(* CODESYS project mpm_fbresult.library
   Title: MPM_FBResult
   Version: 0.0.1.5
   Placeholder: MPM_FBResult
   Company: MatrixPM

Project tree, tasks and I/O mapping:
  data type E_Result
  function block FB_Result_Base [ST]: M_Excute_Ex, M_Execute
  function block FB_ResultBaseITF [ST]: M_Excute_Ex, P_itfResultEx
  function block FB_ResultHelper [ST]: M_MethodResult, P_Result
  function block FB_ResultHelper_V2 [ST]: M_MethodResult
  function block FB_ResultHelper_V2_1 [ST]: M_MethodResult, P_MethodResult
  function block FB_Templete [ST]: M_Execute
  function block FB_Templete_V2 [ST]: M_Execute
  interface ITF_Result: M_Execute
  interface ITF_ResultExtended: _M_Excute
*)

// E_Result
{attribute 'qualified_only'}
TYPE E_Result :
(
	S_OK := 0,
	S_DONE := 1,
	S_FAILED := -1,
	S_WORKING := 3
)DINT;
END_TYPE

// FB_Result_Base
FUNCTION_BLOCK ABSTRACT FB_Result_Base EXTENDS FB_ResultHelper IMPLEMENTS ITF_Result //used to added HRresult to a FB. 
VAR_INPUT
END_VAR
VAR_OUTPUT
END_VAR
VAR
END_VAR

METHOD PROTECTED ABSTRACT M_Excute_Ex : DINT
VAR_INPUT
	lastResult	: DINT;
END_VAR
VAR_INST
END_VAR
END_METHOD

{warning 'add method implementation '}
METHOD FINAL M_Execute : DINT
VAR_INPUT
	lastResult	: DINT;
END_VAR
IF M_MethodResult(M_Execute,lastResult := lastResult) = FALSE THEN
	RETURN;
ELSE
	THIS^.P_Result := THIS^.M_Excute_Ex(THIS^.P_Result);	//FBs implementation
END_IF
END_METHOD

END_FUNCTION_BLOCK

// FB_ResultHelper
(*
Used to implement HRResult style programing to a meathod. This should be implemented inside of a meathod in VAR_INST becuase
this holds state. This should only be used if the meathod won't be able to return the final result in one scan. (async)
*)
FUNCTION_BLOCK FB_ResultHelper //Used to implement HRResult style programing to a meathod. 
VAR_INPUT
END_VAR
VAR_OUTPUT
END_VAR
VAR
	_lastResult			: DINT;		
	pMethodResult		: REFERENCE TO DINT;		
END_VAR
VAR_TEMP
	
END_VAR

METHOD PUBLIC FINAL M_MethodResult : BOOL
VAR_INPUT
	meathodResultRef	: REFERENCE TO DINT;
	lastResult			: DINT;
END_VAR
VAR
END_VAR
VAR_OUTPUT
END_VAR
VAR_INST
END_VAR
IF ADR(meathodResultRef) = 0 THEN
	M_MethodResult := FALSE;	
ELSIF (lastResult > 0 AND (_lastResult = 0 OR _lastResult <> lastResult)) OR ABS(lastResult) = 1 THEN
	meathodResultRef := lastResult;
	M_MethodResult := FALSE;	
ELSIF lastResult = 0 THEN
	pMethodResult REF= meathodResultRef;
	_lastResult := 0;
	M_MethodResult := TRUE;		
ELSE
	pMethodResult REF= meathodResultRef;
	pMethodResult := lastResult;
	M_MethodResult := TRUE;
	_lastResult := lastResult;
END_IF
END_METHOD

PROPERTY PUBLIC P_Result : DINT
GET
IF ADR(pMethodResult) > 0 THEN
	P_Result := pMethodResult;
ELSE
	P_Result := -1; //Maybe 1?
END_IF
END_GET
SET
IF ADR(pMethodResult) > 0 THEN
	_lastResult := P_Result;
	pMethodResult := P_Result;
END_IF
END_SET
END_PROPERTY

END_FUNCTION_BLOCK

// ITF_Result
INTERFACE ITF_Result

METHOD M_Execute : DINT
VAR_INPUT
	lastResult			: DINT;
END_VAR
END_METHOD

END_INTERFACE

// FB_ResultBaseITF
FUNCTION_BLOCK FB_ResultBaseITF EXTENDS FB_Result_Base //used for librays that I can't extened. 
VAR_INPUT
END_VAR
VAR_OUTPUT
END_VAR
VAR
	itfResultEx	: ITF_ResultExtended;
END_VAR

METHOD PROTECTED FINAL M_Excute_Ex : DINT
VAR_INPUT
	lastResult	: DINT;
END_VAR
VAR_INST
END_VAR
IF ADR(itfResultEx) = 0 THEN
	M_Excute_Ex := 1;
	RETURN; 
ELSE
	M_Excute_Ex := itfResultEx._M_Excute(lastResult);
	RETURN; 	
END_IF
END_METHOD

PROPERTY PUBLIC P_itfResultEx : ITF_ResultExtended // has to be set every cycle.
SET
itfResultEx := P_itfResultEx;
END_SET
END_PROPERTY

END_FUNCTION_BLOCK

// ITF_ResultExtended
INTERFACE ITF_ResultExtended EXTENDS ITF_Result

METHOD _M_Excute : DINT //do not call this outside the function
VAR_INPUT
	lastResult	: DINT;
END_VAR
END_METHOD

END_INTERFACE

// FB_ResultHelper_V2
(*
Used to implement HRResult style programing to a meathod. This should be implemented inside of a meathod in VAR_INST becuase
this holds state. This should only be used if the meathod won't be able to return the final result in one scan. (async)
*)
FUNCTION_BLOCK FB_ResultHelper_V2 //Used to implement HRResult style programing to a meathod. 
VAR_INPUT
END_VAR
VAR_OUTPUT
END_VAR
VAR
	_lastResult			: DINT; //stored last result

END_VAR
VAR_TEMP
	
END_VAR

METHOD PUBLIC FINAL M_MethodResult : BOOL
VAR_INPUT
	meathodResultRef	: REFERENCE TO HRESULT; //meathod return
	pMethodResult		: POINTER TO POINTER TO HRESULT; //var to use in meathod calling this		
	lastResult			: HRESULT; //last result passed in through meathod call

END_VAR
VAR
END_VAR
VAR_OUTPUT
END_VAR
VAR_INST
END_VAR
IF ADR(meathodResultRef) = 0 THEN
	M_MethodResult := FALSE;	
ELSIF (lastResult > E_Result.S_OK AND (_lastResult = E_Result.S_OK OR _lastResult <> lastResult)) OR ABS(lastResult) = 1 THEN //dont run
	meathodResultRef := lastResult;
	M_MethodResult := FALSE;	
ELSIF lastResult = E_Result.S_OK THEN //reset so run
	pMethodResult^ := ADR(meathodResultRef);
	_lastResult := 0;
	M_MethodResult := TRUE;		
ELSE //working
	pMethodResult^ := ADR(meathodResultRef);
	pMethodResult^^ := lastResult;
	M_MethodResult := TRUE;
	_lastResult := lastResult;
END_IF
END_METHOD

END_FUNCTION_BLOCK

// FB_ResultHelper_V2_1
(*
Used to implement HRResult style programing to a meathod. This should be implemented inside of a meathod in VAR_INST becuase
this holds state. This should only be used if the meathod won't be able to return the final result in one scan. (async)
*)
FUNCTION_BLOCK FB_ResultHelper_V2_1 //Used to implement HRResult style programing to a meathod. 
VAR_INPUT
END_VAR
VAR_OUTPUT
END_VAR
VAR
	_lastResult			: POINTER TO HRESULT; //stored last result	
	meathodResultRef	: REFERENCE TO HRESULT; //meathod return
END_VAR
VAR_TEMP
	
END_VAR

METHOD PUBLIC FINAL M_MethodResult : BOOL
VAR_INPUT
	meathodResultRef	: REFERENCE TO HRESULT; //meathod return
	lastResult			: HRESULT; //last result passed in through meathod call
	_lastResult			: POINTER TO HRESULT; //stored last result	
END_VAR
VAR
END_VAR
VAR_OUTPUT
END_VAR
VAR_INST
END_VAR
THIS^._lastResult := _lastResult;
THIS^.meathodResultRef REF= meathodResultRef;
IF ADR(meathodResultRef) = 0 THEN
	M_MethodResult := FALSE;	
ELSIF (ABS(lastResult) = 1) THEN // IS LAST RESULT IS DONE OR FAILED 
	meathodResultRef := lastResult; //RETURN LASTRESULT
	M_MethodResult := FALSE;		
ELSIF (lastResult > E_Result.S_DONE AND //WORKING PASS LAST RESULT BACK UP AS IS
	_lastResult^ = E_Result.S_OK) THEN //LAST RESULT WAS OK
	meathodResultRef := lastResult; //RETURN LASTRESULT
	M_MethodResult := FALSE;	
ELSIF (lastResult > E_Result.S_DONE	AND _lastResult^ = lastResult) THEN //WORKING LAST RESULT and matching
	meathodResultRef := _lastResult^; //RETURN STORED LASTRESULT
	M_MethodResult := TRUE;	
ELSIF (lastResult > E_Result.S_DONE	AND _lastResult^ <> lastResult) THEN //WORKING LAST RESULT and not matching
	meathodResultRef := _lastResult^; //RETURN STORED LASTRESULT
	M_MethodResult := FALSE;		
ELSIF lastResult = E_Result.S_OK THEN //reset so run
	_lastResult^ := 0;
	M_MethodResult := TRUE;		
ELSE //working
	M_MethodResult := TRUE;
	_lastResult^ := lastResult;
END_IF
END_METHOD

PROPERTY P_MethodResult : HResult
GET
P_MethodResult := meathodResultRef;
END_GET
SET
meathodResultRef := P_MethodResult;
_lastResult^ := P_MethodResult;
END_SET
END_PROPERTY

END_FUNCTION_BLOCK

// FB_Templete
FUNCTION_BLOCK ABSTRACT FB_Templete //DO NOT IMPLMENT
VAR_INPUT
END_VAR
VAR_OUTPUT
END_VAR
VAR
END_VAR

//This a templete for implentating helper

METHOD M_Execute : DINT
VAR_INPUT
	lastResult : DINT;
END_VAR
VAR
	_state			: DINT;
	_fbResult		: FB_ResultHelper;
END_VAR
//This a templete for implentation

IF _fbResult.M_MethodResult(M_Execute,lastResult) = FALSE THEN
	RETURN;
ELSE	
	IF lastResult = E_Result.S_OK THEN //Reset
		_state := 0;	
	END_IF 	
	
	_fbResult.P_Result := E_Result.S_WORKING; //Working	
	
	CASE _state OF
		0:
		
	END_CASE

END_IF
END_METHOD

END_FUNCTION_BLOCK

// FB_Templete_V2
FUNCTION_BLOCK ABSTRACT FB_Templete_V2 //DO NOT IMPLMENT
VAR_INPUT
END_VAR
VAR_OUTPUT
END_VAR
VAR
END_VAR

//This a templete for implentating helper

METHOD M_Execute : HRESULT
VAR_INPUT
	lastResult : DINT;
END_VAR
VAR
	_state			: DINT;
	_fbResult		: FB_ResultHelper_V2;
	pResult : REFERENCE TO HRESULT;
END_VAR
//This a templete for implentation

IF _fbResult.M_MethodResult(M_Execute,pResult,lastResult) = FALSE THEN
	RETURN;
ELSE	
	IF pResult = E_Result.S_OK THEN //Reset
		_state := 0;	
	END_IF 	
	
	pResult := E_Result.S_WORKING; //Working	
	
	CASE _state OF
		0:
		
	END_CASE

END_IF
END_METHOD

END_FUNCTION_BLOCK
